(* PLC project Unnamed, Unknown Unnamed 1 *)
(* stored: creationDateTime 2025-10-10T14:27:24, modificationDateTime 2025-10-10T17:02:34 *)

PROGRAM rd_seq_rbear_trap
  VAR
    RANDOM : UINT;
    SEED : UINT := 123;
    A : UINT := 123;
    C : UINT := 123;
    M : UINT := 123;
    DISPLAY : UINT;
  END_VAR
  VAR  (* added by the conversion: wires and edge detectors of the diagram *)
    _MUL1_OUT : UINT;
  END_VAR

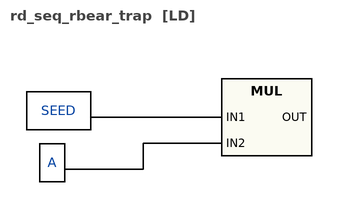
(* LD diagram, written out as Structured Text *)
_MUL1_OUT := SEED * A;
END_PROGRAM

CONFIGURATION Config0
  RESOURCE Res0 ON PLC
    TASK task0(INTERVAL := T#20ms, PRIORITY := 0);
    PROGRAM instance0 WITH task0 : rd_seq_rbear_trap;
  END_RESOURCE
END_CONFIGURATION
